TYPE ST_CYIo ://气缸 I O
STRUCT
	DIOnSwitch:		    BOOL;	//开限位
	DIOFFSwitch:		BOOL;	//关限位

	DOStatus1:          BOOL;//输出状态
	DOStatus2:          BOOL;//输出状态

END_STRUCT
END_TYPE

(* stored: Version 1.1.0.1, ProductVersion 3.1.4024.9
   DUT ST_CYIo: Id {9b476a03-796e-4a84-98b0-5d15e563a978} *)
